Staubli VAL3: Refresh3.pgx

program Refresh3()
begin
  //选择工具/坐标系界面
  if bUserRefresh
    cls()
    userPage()
    gotoxy(1,1)
    put("F1->确定")
    gotoxy(1,13)
    put("F1")
    gotoxy(1,2)
    put("F2->编辑")
    gotoxy(6,13)
    put("F2")
//    gotoxy(1,3)
//    put("F3->删除")
//    gotoxy(11,13)
//    put("F3")
//    gotoxy(1,4)
//    put("F4->选择工具/坐标系")
//    gotoxy(16,13)
//    put("F4")
    //
//    gotoxy(1,6)
//    put("F6->")
//    gotoxy(26,13)
//    put("")
    gotoxy(1,7)
    put("F7->保存")
    gotoxy(31,13)
    put("F7")
    gotoxy(1,8)
    put("F8->返回")
    gotoxy(36,13)
    put("F8")
  endIf
end
